(* PLC project tri_chain, Dassault Systèmes ControlBuild 2024x *)
(* stored: creationDateTime 2023-10-03T11:13:58-01:00 *)

PROGRAM tri_chain.tri_chain

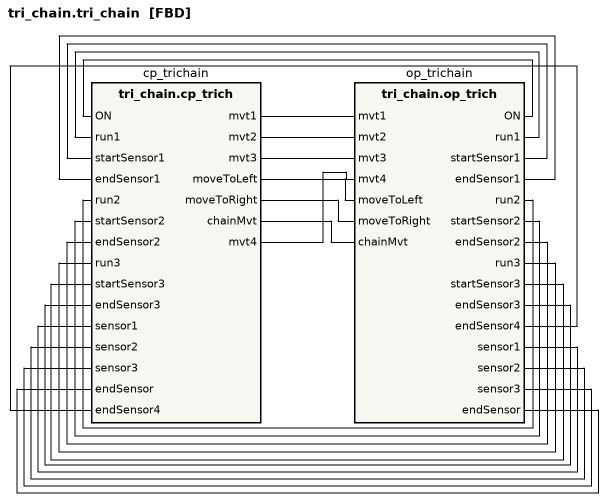
(* FBD diagram, written out as Structured Text *)
op_trichain(mvt1 := cp_trichain.mvt1, mvt2 := cp_trichain.mvt2, mvt3 := cp_trichain.mvt3, mvt4 := cp_trichain.mvt4, moveToLeft := cp_trichain.moveToLeft, moveToRight := cp_trichain.moveToRight, chainMvt := cp_trichain.chainMvt);
cp_trichain(ON := op_trichain.ON, run1 := op_trichain.run1, startSensor1 := op_trichain.startSensor1, endSensor1 := op_trichain.endSensor1, run2 := op_trichain.run2, startSensor2 := op_trichain.startSensor2, endSensor2 := op_trichain.endSensor2, run3 := op_trichain.run3, startSensor3 := op_trichain.startSensor3, endSensor3 := op_trichain.endSensor3, sensor1 := op_trichain.sensor1, sensor2 := op_trichain.sensor2, sensor3 := op_trichain.sensor3, endSensor := op_trichain.endSensor, endSensor4 := op_trichain.endSensor4);
END_PROGRAM
